PROGRAM prgKNX
VAR
	fbKBusState				: FB_K_Bus_State;
	fbKNXMaster				: FB_KL6301_KNX_Master;
	fbRampHeating			: FB_OBC_OnOff_KNX;				//{#lynus.ag#()}
	fbTreeHeating			: FB_OBC_OnOff_KNX;				//{#lynus.ag#()}
	fbPumpFishSea			: FB_OBC_OnOff_KNX;				//{#lynus.ag#()}
	fbPumpSwimSea			: FB_OBC_OnOff_KNX;				//{#lynus.ag#()}
	bOnEmergPowerOffRH		: BOOL;							//{#lynus.ag#()}
	bOnEmergPowerOffTH		: BOOL;							//{#lynus.ag#()}
	bOnEmergPowerOffPFish	: BOOL;							//{#lynus.ag#()}
	bOnEmergPowerOffPSwim	: BOOL;							//{#lynus.ag#()}
	bSOnEmergPowerOffRH		: BOOL;							//{#lynus.ag#()}
	bSOnEmergPowerOffTH		: BOOL;							//{#lynus.ag#()}
	bSOnEmergPowerOffPFish	: BOOL;							//{#lynus.ag#()}
	bSOnEmergPowerOffPSwim	: BOOL;							//{#lynus.ag#()}
	byErrorWarningRH		: BYTE;							//{#lynus.ag#()}
	byErrorWarningTH		: BYTE;							//{#lynus.ag#()}
	byErrorWarningPFish		: BYTE;							//{#lynus.ag#()}
	byErrorWarningPSwim		: BYTE;							//{#lynus.ag#()}
END_VAR

//Power Data
//Ramp Heating 34kw
//Three Heating 13kW 
//Fish Sea pump 7.5kW
//Swim Sea Pump 7.5kw

//K-Bus State
fbKBusState(uiKBusState_OUT=> );

//Configure the KXN Master
fbKNXMaster.stPhysAddrTerminal.Area := 1;
	fbKNXMaster.stPhysAddrTerminal.Device := 160;
		fbKNXMaster.stPhysAddrTerminal.Line := 9;
		
fbKNXMaster.arrGroupFilter[1].GROUP_ADDR.MAIN := 6;
	fbKNXMaster.arrGroupFilter[1].GROUP_ADDR.NUMBER := 0;
		fbKNXMaster.arrGroupFilter[1].GROUP_ADDR.SUB_MAIN := 1;
fbKNXMaster.arrGroupFilter[1].GROUP_LEN := 4;	
	
fbKNXMaster(
	stPhysAddrTerminal:= , 
	arrGroupFilter:= , 
	iKL6301Mode:= 0, 
	uiKBusState_IN:= fbKBusState.uiKBusState_OUT, 
	bActive=> , 
	bReady=> , 
	byErrorWarning=> , 
	diNrOfKNXMasterLine_OUT=> , 
	eMessageKNXMaster=> );

fbTreeHeating.strGroupAddr.MAIN := 6;
	fbTreeHeating.strGroupAddr.SUB_MAIN := 1;
		fbTreeHeating.strGroupAddr.NUMBER := 0;	

fbTreeHeating.stSetupOBC.bOnEmergPowerOff := bOnEmergPowerOffTH;
	
fbTreeHeating(
	bEnable:= , 
	bPowerDataInvers:= , 
	diNrOfKNXMasterLine_IN:= fbKNXMaster.diNrOfKNXMasterLine_OUT, 
	diNrOfEMS_IN:= prgEMS.EMS.diNrOfEMS_OUT, 
	diNrOfEM_IN_OBC:= , 
	stSetupOBC:= , 
	strGroupAddr:= , 
	stDataOBC=> , 
	diNrOfOBC_OUT=> );

byErrorWarningTH := fbTreeHeating.stDataOBC.byErrorWarning;	
	bSOnEmergPowerOffTH := fbTreeHeating.stDataOBC.bSOnEmergPowerOff;	
	
fbPumpFishSea.strGroupAddr.MAIN := 6;
	fbPumpFishSea.strGroupAddr.SUB_MAIN := 1;
		fbPumpFishSea.strGroupAddr.NUMBER := 2;	

fbPumpFishSea.stSetupOBC.bOnEmergPowerOff := bOnEmergPowerOffPFish;
	
fbPumpFishSea(
	bEnable:= , 
	bPowerDataInvers:= , 
	diNrOfKNXMasterLine_IN:= fbKNXMaster.diNrOfKNXMasterLine_OUT, 
	diNrOfEMS_IN:= prgEMS.EMS.diNrOfEMS_OUT, 
	diNrOfEM_IN_OBC:= , 
	stSetupOBC:= , 
	strGroupAddr:= , 
	stDataOBC=> , 
	diNrOfOBC_OUT=> );

byErrorWarningPFish := fbPumpFishSea.stDataOBC.byErrorWarning;
	bSOnEmergPowerOffPFish := fbPumpFishSea.stDataOBC.bSOnEmergPowerOff;		
	
fbPumpSwimSea.strGroupAddr.MAIN := 6;
	fbPumpSwimSea.strGroupAddr.SUB_MAIN := 1;
		fbPumpSwimSea.strGroupAddr.NUMBER := 3;	

fbPumpSwimSea.stSetupOBC.bOnEmergPowerOff := bOnEmergPowerOffPSwim;
	
fbPumpSwimSea(
	bEnable:= , 
	bPowerDataInvers:= , 
	diNrOfKNXMasterLine_IN:= fbKNXMaster.diNrOfKNXMasterLine_OUT, 
	diNrOfEMS_IN:= prgEMS.EMS.diNrOfEMS_OUT, 
	diNrOfEM_IN_OBC:= , 
	stSetupOBC:= , 
	strGroupAddr:= , 
	stDataOBC=> , 
	diNrOfOBC_OUT=> );

byErrorWarningPSwim := fbPumpSwimSea.stDataOBC.byErrorWarning;	
	bSOnEmergPowerOffPSwim := fbPumpSwimSea.stDataOBC.bSOnEmergPowerOff;
	
fbRampHeating.strGroupAddr.MAIN := 6;
	fbRampHeating.strGroupAddr.SUB_MAIN := 1;
		fbRampHeating.strGroupAddr.NUMBER := 1;	

fbRampHeating.stSetupOBC.bOnEmergPowerOff := bOnEmergPowerOffRH;
	
fbRampHeating(
	bEnable:= , 
	bPowerDataInvers:= , 
	diNrOfKNXMasterLine_IN:= fbKNXMaster.diNrOfKNXMasterLine_OUT, 
	diNrOfEMS_IN:= prgEMS.EMS.diNrOfEMS_OUT, 
	diNrOfEM_IN_OBC:= , 
	stSetupOBC:= , 
	strGroupAddr:= , 
	stDataOBC=> , 
	diNrOfOBC_OUT=> );
	
byErrorWarningRH := fbRampHeating.stDataOBC.byErrorWarning;	
	bSOnEmergPowerOffRH := fbRampHeating.stDataOBC.bSOnEmergPowerOff;

END_PROGRAM

(* stored: Version 1.1.0.1, ProductVersion 3.1.4024.9
   POU prgKNX: Id {27734d39-760d-47bd-8318-923a7873e7e1}, SpecialFunc None *)
